Fanuc KAREL source: V_OVERRIDE.kl

PROGRAM T
%NOLOCKGROUP
VAR
 v0 : STRING[40]
 v1 : REAL
 v2 : INTEGER
BEGIN
 V_OVERRIDE(v0, v1, v2)
END T
